{attribute 'qualified_only'}
{attribute 'to_string'}
{attribute 'strict'}
TYPE E_INSTANCE_CMD : // instructions for fb_Instance executions
(
	NULL,
  INIT,
  DISABLE,
  ENABLE,
  WORK,
  PROCEED := 100,
  FINISH,
  CLEAR
)UINT;
END_TYPE

(* stored: Version 1.1.0.1, ProductVersion 3.1.4026.18
   DUT E_INSTANCE_CMD: Id {0fe500de-a497-4dc5-927c-5fead3ff445e} *)
